FUNCTION "HLP_BitPutGet" : Void
{ S7_Optimized_Access := 'TRUE' }
VERSION : 0.1
   VAR_INPUT
      iSR : Bool;   // TRUE - S, FALSE - R
      iBitNr : Variant;
   END_VAR

   VAR_IN_OUT
      ioValue : Variant;
   END_VAR


BEGIN
END_FUNCTION

